FUNCTION_BLOCK FB_CFC_SamplePouPageOriented
VAR_INPUT
//	eOperation	: INT;
	eOperation	: E_Operation;
END_VAR
VAR_OUTPUT
	iResultC	: DINT;
END_VAR
VAR
	arrDataA	: ARRAY [1..iMax] OF DINT;
	arrDataB	: ARRAY [1..iMax] OF DINT;
	arrDataC	: ARRAY [1..iMax] OF DINT;
	I 			: DINT;
	bInit		: BOOL := TRUE;
END_VAR
VAR CONSTANT
	iMax 		: DINT := 10;
END_VAR
VAR // added by the converter: edge detectors and wires of the graphical bodies
    _w1, _w2, _w4, _w6, _w10 : DINT;
    _w3, _w5, _w9 : ANY;
    _w7, _w8 : BOOL;
END_VAR


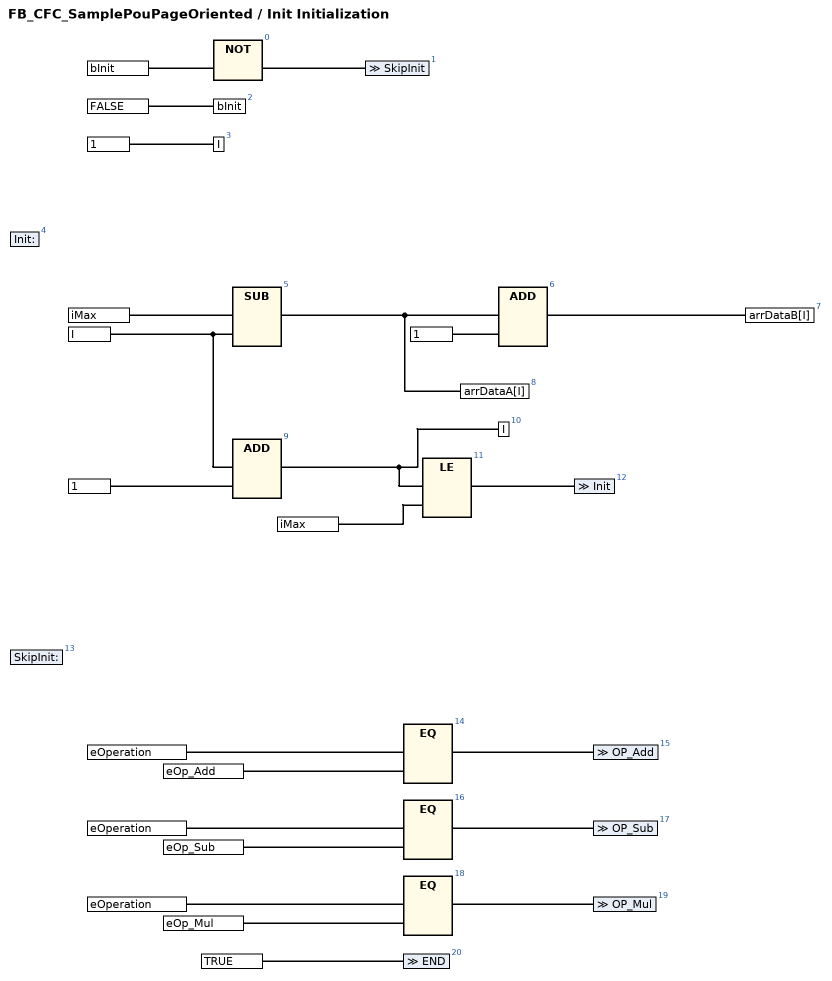
// PAGE Init Initialization
IF NOT bInit THEN JMP SkipInit; END_IF
bInit := FALSE;
I := 1;
Init: ;
_w1 := iMax - I;
arrDataB[I] := _w1 + 1;
arrDataA[I] := _w1;
_w2 := I + 1;
I := _w2;
IF _w2 <= iMax THEN JMP Init; END_IF
SkipInit: ;
IF eOperation = eOp_Add THEN JMP OP_Add; END_IF
IF eOperation = eOp_Sub THEN JMP OP_Sub; END_IF
IF eOperation = eOp_Mul THEN JMP OP_Mul; END_IF
IF TRUE THEN JMP END; END_IF

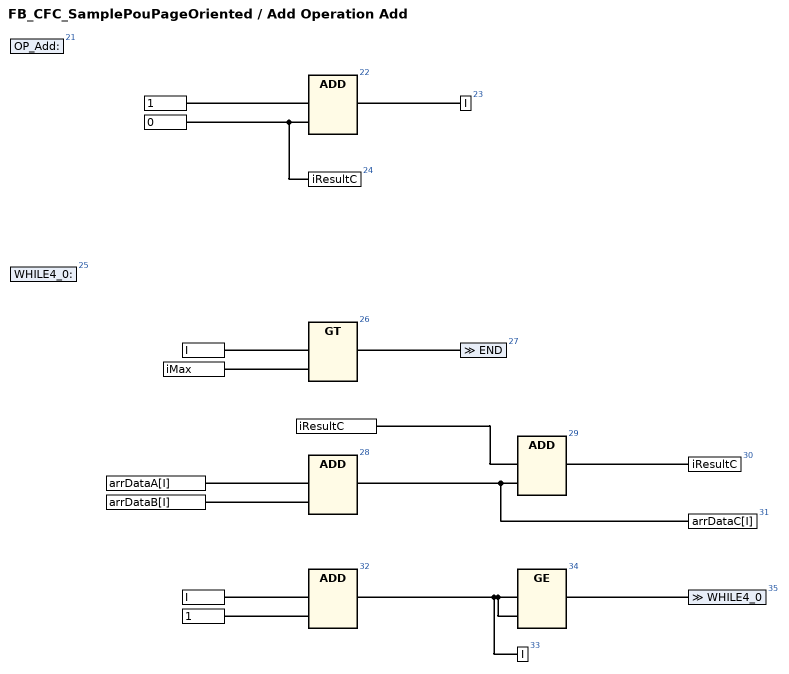
// PAGE Add Operation Add
OP_Add: ;
I := 1 + 0;
iResultC := 0;
WHILE4_0: ;
IF I > iMax THEN JMP END; END_IF
_w3 := arrDataA[I] + arrDataB[I];
iResultC := iResultC + _w3;
arrDataC[I] := _w3;
_w4 := I + 1;
I := _w4;
IF _w4 >= _w4 THEN JMP WHILE4_0; END_IF

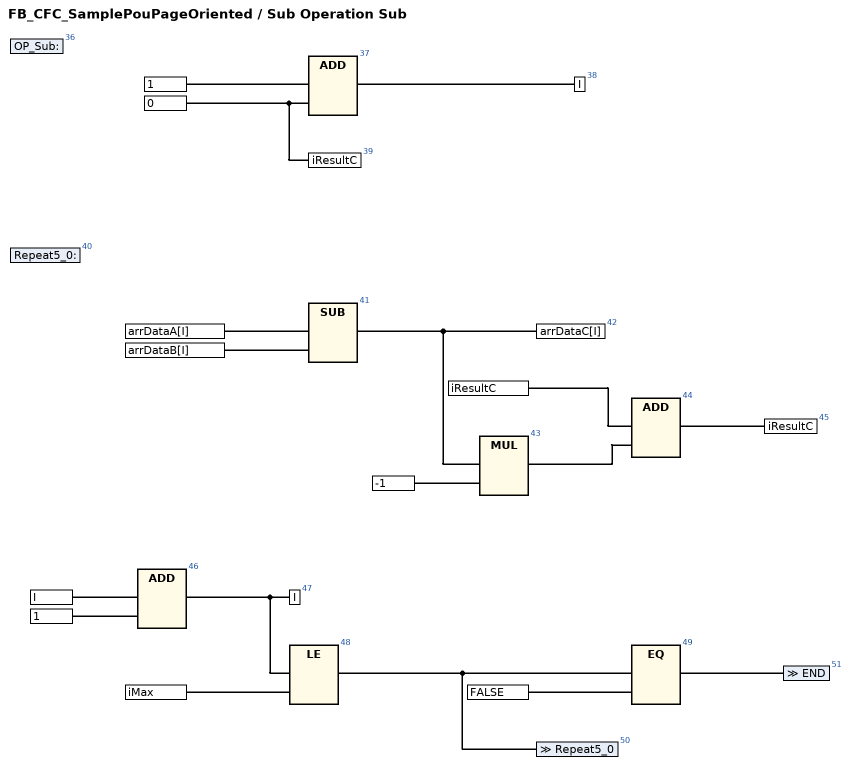
// PAGE Sub Operation Sub
OP_Sub: ;
I := 1 + 0;
iResultC := 0;
Repeat5_0: ;
_w5 := arrDataA[I] - arrDataB[I];
arrDataC[I] := _w5;
iResultC := iResultC + _w5 * -1;
_w6 := I + 1;
I := _w6;
_w7 := _w6 <= iMax;
_w8 := _w7 = FALSE;
IF _w7 THEN JMP Repeat5_0; END_IF
IF _w8 THEN JMP END; END_IF

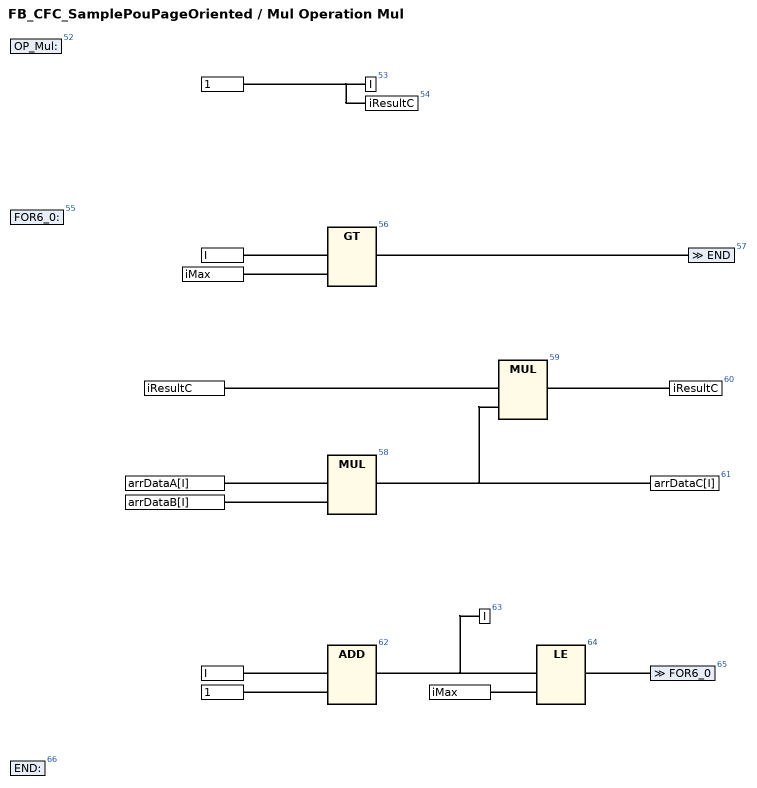
// PAGE Mul Operation Mul
OP_Mul: ;
I := 1;
iResultC := 1;
FOR6_0: ;
IF I > iMax THEN JMP END; END_IF
_w9 := arrDataA[I] * arrDataB[I];
iResultC := iResultC * _w9;
arrDataC[I] := _w9;
_w10 := I + 1;
I := _w10;
IF _w10 <= iMax THEN JMP FOR6_0; END_IF
END: ;

END_FUNCTION_BLOCK

(* stored: Version 1.1.0.1, ProductVersion 3.1.4024.11
   POU FB_CFC_SamplePouPageOriented: Id {152d40ab-bdb6-4a7d-b84a-962b022c485e}, SpecialFunc None *)
